// TwinCAT 3 PLC project AutoWarehouseSort
// ProgramVersion: 3.1.4024.0
// libraries:
//   Tc2_Standard, * (Beckhoff Automation GmbH)
//   Tc2_System, * (Beckhoff Automation GmbH)
//   Tc3_EventLogger, * (Beckhoff Automation GmbH)
//   Tc3_Module, * (Beckhoff Automation GmbH)
// project tree:
//   DUTs/ eMotorStates.TcDUT
//   / PlcTask.TcTTO
//   POUs/ AlarmWithCustomSourceInfo.TcPOU, MAIN.TcPOU, ConfirmableAlarmWithArguments.TcPOU
//   POUs/Devices/Motors/ conveyorMotor.TcPOU
//   POUs/Interfaces/ Imotor.TcIO
// real-time tasks:
//   TASK PlcTask: cycle T#10ms, priority 20, ADS port 350

CONFIGURATION AutoWarehouseSort
    RESOURCE PLC ON TwinCAT3
        TASK PlcTask(INTERVAL := T#10ms, PRIORITY := 20);
        PROGRAM MAIN WITH PlcTask : MAIN;
        PROGRAM ConfirmableAlarmWithArguments WITH PlcTask : ConfirmableAlarmWithArguments;
        PROGRAM AlarmWithCustomSourceInfo WITH PlcTask : AlarmWithCustomSourceInfo;
    END_RESOURCE
END_CONFIGURATION

// ---- DUTs/eMotorStates.TcDUT
{attribute 'qualified_only'}
{attribute 'strict'}
TYPE eMotorStates :
(
	firstrun, running, stopped, errored, starting, stopping, pause, paused
);
END_TYPE

// ---- POUs/Interfaces/Imotor.TcIO
INTERFACE Imotor

PROPERTY error : bool
GET
END_GET
SET
END_SET
END_PROPERTY

METHOD run : BOOL
END_METHOD

PROPERTY running : bool
GET
END_GET
SET
END_SET
END_PROPERTY

METHOD status : BOOL
END_METHOD

METHOD stop : BOOL
VAR_INPUT
END_VAR
END_METHOD

END_INTERFACE

// ---- POUs/MAIN.TcPOU
PROGRAM MAIN
VAR
    bInit : BOOL := TRUE; 
    bSend : BOOL := TRUE; 

    fbMsg : FB_TcMessage; 
	conveyorMotor1 : conveyorMotor;
END_VAR

IF bInit THEN
	bInit := FALSE;
	fbMsg.CreateEx(TC_Events.AlarmsAndEvents.Estop, 0);
END_IF

IF bSend THEN
	bSend := FALSE;
	fbMsg.Send(0);
	
END_IF

END_PROGRAM

// ---- POUs/Devices/Motors/conveyorMotor.TcPOU
FUNCTION_BLOCK conveyorMotor IMPLEMENTS Imotor
VAR_INPUT
END_VAR
VAR_OUTPUT
END_VAR
VAR
	bStartMotor : BOOL := FALSE;
	bStopMotor : BOOL := TRUE;
	bPauseMotor : BOOL := FALSE;
	eStates : eMotorStates := eMotorStates.firstrun;
	isMotorRunning : BOOL :=  FALSE;
	isError : BOOL := FALSE;
END_VAR

CASE eStates OF
	eMotorStates.firstrun :
		IF bStartMotor THEN
			eStates := eMotorStates.starting;
		END_IF
	eMotorStates.starting:
		IF NOT bStopMotor THEN
			run();
			eStates := eMotorStates.running;
			isMotorRunning := TRUE;
		END_IF
	eMotorStates.running:
		IF bStopMotor THEN
			stop();
			isMotorRunning := FALSE;	
			eStates := eMotorStates.stopped;
		END_IF
		IF bPauseMotor THEN
			eStates := eMotorStates.pause;
		END_IF
	eMotorStates.stopped:
		IF bStartMotor AND NOT bStopMotor THEN
			eStates := eMotorStates.running;
		END_IF
	eMotorStates.pause:
		MpauseMotor();
		eStates := eMotorStates.paused;
	eMotorStates.paused:
		IF bStartMotor AND NOT bStopMotor THEN
			eStates := eMotorStates.running;
		END_IF
		IF  bStopMotor THEN
			eStates := eMotorStates.stopping;
		END_IF
END_CASE


PROPERTY error : BOOL
GET
VAR
	bError : BOOL;
END_VAR
error := isError;
END_GET
SET
isError := error;
END_SET
END_PROPERTY

METHOD MpauseMotor : BOOL
VAR_INPUT
END_VAR
END_METHOD

METHOD run : BOOL
VAR
	bRunMotor: BOOL;
END_VAR
bRunMotor := TRUE;
END_METHOD


PROPERTY running : BOOL
GET
running := isMotorRunning;
END_GET
SET
VAR
	bSimRun : BOOL := False;
END_VAR
isMotorRunning := running;
END_SET
END_PROPERTY

METHOD status : BOOL
VAR
	fbAlarm	: Tc3_EventLogger.FB_TcAlarm;
	bRaiseAlarm	: BOOL;
	bClearAlarm	: BOOL;
	bConfirmAlarm	: BOOL;
	fbSourceInfo	: Tc3_EventLogger.FB_TcSourceInfo;
END_VAR
bRaiseAlarm := TRUE;
END_METHOD

METHOD stop : BOOL
VAR
	bStopM : BOOL;
END_VAR
bStopM := TRUE;
END_METHOD

END_FUNCTION_BLOCK

// ---- POUs/ConfirmableAlarmWithArguments.TcPOU
PROGRAM ConfirmableAlarmWithArguments
VAR
	bIsInitialized : BOOL;
	fbAlarm : FB_TcAlarm;
	bRaiseAlarm : BOOL;
	bClearAlarm : BOOL;
	bConfirmAlarm : BOOL;
END_VAR

IF NOT bIsInitialized THEN
	bIsInitialized := TRUE;
	fbAlarm.CreateEx(TC_Events.AlarmsAndEvents.Stop, TRUE, 0);
END_IF

IF bRaiseAlarm THEN
	bRaiseAlarm := FALSE;
	fbAlarm.ipArguments.Clear().AddString('Alice');
	fbAlarm.Raise(0);
END_IF

IF bConfirmAlarm THEN
	bConfirmAlarm := FALSE;
	fbAlarm.Confirm(0);
END_IF

IF bClearAlarm THEN
	bClearAlarm := FALSE;
	fbAlarm.Clear(0, FALSE);
END_IF

END_PROGRAM

// ---- POUs/AlarmWithCustomSourceInfo.TcPOU
PROGRAM AlarmWithCustomSourceInfo
VAR
	bIsInitalized : BOOL;
    fbAlarm : FB_TcAlarm;
    bRaiseAlarm : BOOL;
    bClearAlarm : BOOL;
    fbSourceInfo : FB_TcSourceInfo;
END_VAR

IF NOT bIsInitalized THEN
    bIsInitalized := TRUE;
    fbSourceInfo.Clear();
    fbSourceInfo.sName := 'Water pump 3';
    fbAlarm.CreateEx(TC_Events.AlarmsAndEvents.Stop, FALSE, fbSourceInfo);
END_IF

IF bRaiseAlarm THEN
    bRaiseAlarm := FALSE;
    fbAlarm.ipArguments.Clear().AddString('Bob');
    fbAlarm.Raise(0);
END_IF

IF bClearAlarm THEN
    bClearAlarm := FALSE;
    fbAlarm.Clear(0, TRUE);
END_IF

END_PROGRAM
